% RSLogix 500 project P3_KOBIERSKI_M.RSS, saved by version 8.30.00.16 %
PROJECT "UNTITLED"    % processor: Bul.1763 MicroLogix 1100 Series B %

PROGRAM FILES
  LAD 2 "MAIN"  3 rungs
  LAD 3 "CLEAN SCAN"  6 rungs
  LAD 4 "INCOMING"  4 rungs
  LAD 5 "OUTGOING"  4 rungs

DATA FILES
  O0 OUTPUT  4 elements
  I1 INPUT  6 elements
  S2 STATUS  66 elements
  B3 BINARY  1 elements
  T4 TIMER  1 elements
  C5 COUNTER  1 elements
  R6 CONTROL  1 elements
  N7 INTEGER  6 elements
  F8 FLOAT  1 elements
  ST9 SCAN  6 elements

LADDER 2 "MAIN"
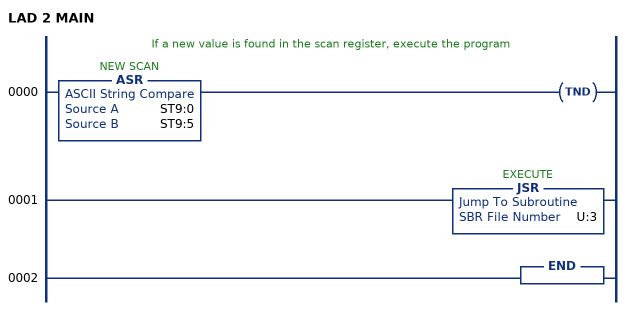
% Rung: 0 %
% If a new value is found in the scan register, execute the program %
SOR ASR ST9:0 ST9:5 TND EOR
%   ST9:0  "NEW SCAN" %
%   ST9:5  "ZERO" %
% Rung: 1 %
SOR JSR U:3 EOR
%   U:3  "EXECUTE" %
% Rung: 2 %
SOR END EOR

LADDER 3 "CLEAN SCAN"
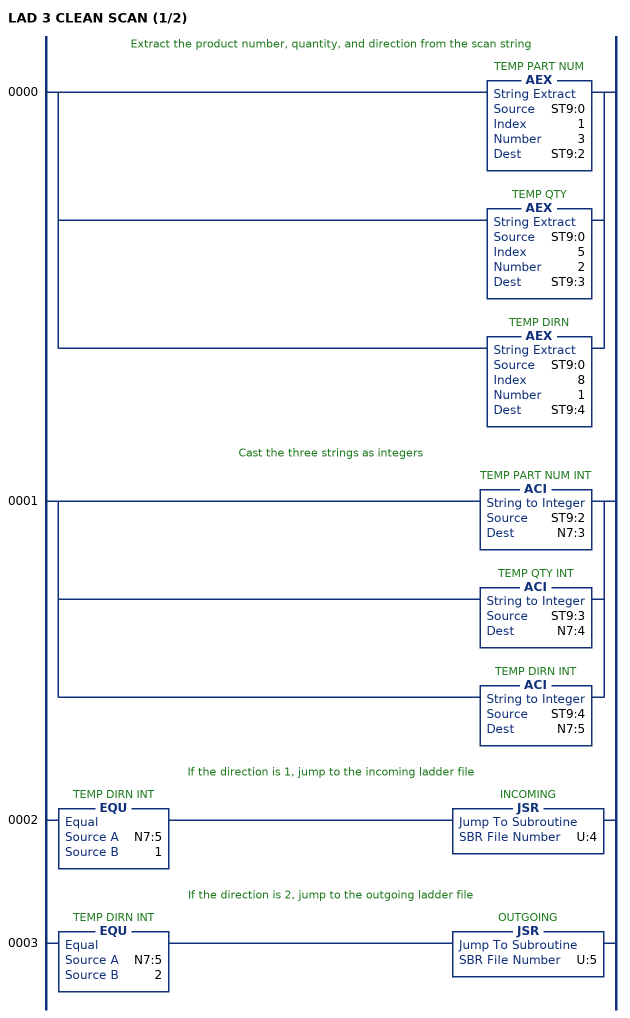
% Rung: 0 %
% Extract the product number, quantity, and direction from the scan string %
SOR BST AEX ST9:0 1 3 ST9:2 NXB AEX ST9:0 5 2 ST9:3 NXB AEX ST9:0 8 1 ST9:4 BND EOR
%   ST9:0  "NEW SCAN" %
%   ST9:2  "TEMP PART NUM" %
%   ST9:3  "TEMP QTY" %
%   ST9:4  "TEMP DIRN" %
% Rung: 1 %
% Cast the three strings as integers %
SOR BST ACI ST9:2 N7:3 NXB ACI ST9:3 N7:4 NXB ACI ST9:4 N7:5 BND EOR
%   ST9:2  "TEMP PART NUM" %
%   N7:3  "TEMP PART NUM INT" %
%   ST9:3  "TEMP QTY" %
%   N7:4  "TEMP QTY INT" %
%   ST9:4  "TEMP DIRN" %
%   N7:5  "TEMP DIRN INT" %
% Rung: 2 %
% If the direction is 1, jump to the incoming ladder file %
SOR EQU N7:5 1 JSR U:4 EOR
%   N7:5  "TEMP DIRN INT" %
%   U:4  "INCOMING" %
% Rung: 3 %
% If the direction is 2, jump to the outgoing ladder file %
SOR EQU N7:5 2 JSR U:5 EOR
%   N7:5  "TEMP DIRN INT" %
%   U:5  "OUTGOING" %

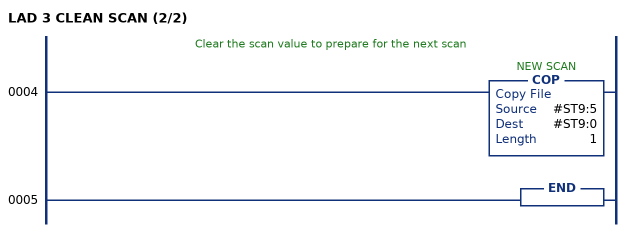
% Rung: 4 %
% Clear the scan value to prepare for the next scan %
SOR COP #ST9:5 #ST9:0 1 EOR
%   ST9:5  "ZERO" %
%   ST9:0  "NEW SCAN" %
% Rung: 5 %
SOR END EOR

LADDER 4 "INCOMING"
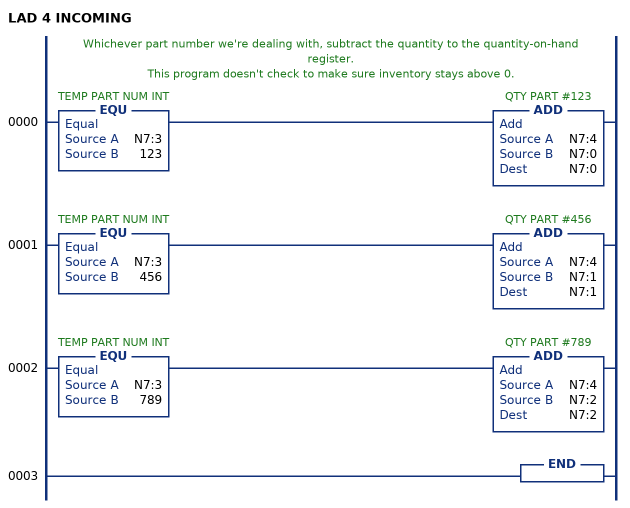
% Rung: 0 %
% Whichever part number we're dealing with, subtract the quantity to the quantity-on-hand register.
% This program doesn't check to make sure inventory stays above 0. %
SOR EQU N7:3 123 ADD N7:4 N7:0 N7:0 EOR
%   N7:3  "TEMP PART NUM INT" %
%   N7:4  "TEMP QTY INT" %
%   N7:0  "QTY PART #123" %
% Rung: 1 %
SOR EQU N7:3 456 ADD N7:4 N7:1 N7:1 EOR
%   N7:3  "TEMP PART NUM INT" %
%   N7:4  "TEMP QTY INT" %
%   N7:1  "QTY PART #456" %
% Rung: 2 %
SOR EQU N7:3 789 ADD N7:4 N7:2 N7:2 EOR
%   N7:3  "TEMP PART NUM INT" %
%   N7:4  "TEMP QTY INT" %
%   N7:2  "QTY PART #789" %
% Rung: 3 %
SOR END EOR

LADDER 5 "OUTGOING"
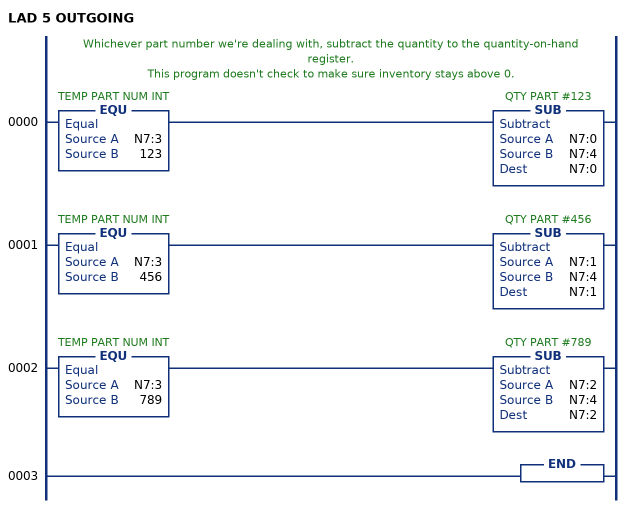
% Rung: 0 %
% Whichever part number we're dealing with, subtract the quantity to the quantity-on-hand register.
% This program doesn't check to make sure inventory stays above 0. %
SOR EQU N7:3 123 SUB N7:0 N7:4 N7:0 EOR
%   N7:3  "TEMP PART NUM INT" %
%   N7:0  "QTY PART #123" %
%   N7:4  "TEMP QTY INT" %
% Rung: 1 %
SOR EQU N7:3 456 SUB N7:1 N7:4 N7:1 EOR
%   N7:3  "TEMP PART NUM INT" %
%   N7:1  "QTY PART #456" %
%   N7:4  "TEMP QTY INT" %
% Rung: 2 %
SOR EQU N7:3 789 SUB N7:2 N7:4 N7:2 EOR
%   N7:3  "TEMP PART NUM INT" %
%   N7:2  "QTY PART #789" %
%   N7:4  "TEMP QTY INT" %
% Rung: 3 %
SOR END EOR

OTHER DOCUMENTED ADDRESSES
  B3:0/0  "EXECUTE"
  N7:0/3  "HOLDOVER INT"
  ST9:0.0  "NEW SCAN"
  ST9:1  "OLD SCAN"

DATA TABLE (non-zero values as saved)
DATA ST9
% ST9:0 % "0"
% ST9:2 % "0"
% ST9:3 % "0"
% ST9:4 % "0"
